TYPE AxisInfo :
STRUCT
	openPosition: LREAL;
	closedPosition: LREAL;
END_STRUCT
END_TYPE

(* stored: Version 1.1.0.1, ProductVersion 3.1.4020.12
   DUT AxisInfo: Id {e58a7f0c-7853-4f34-a842-3b9873755760} *)
